FUNCTION_BLOCK TEMPLATE_NEURALFB
  (* Standard: 61499-2 *)
  (* Version 1.0, 11-01-12, GASR, Universidade do Estado de Santa Catarina *)
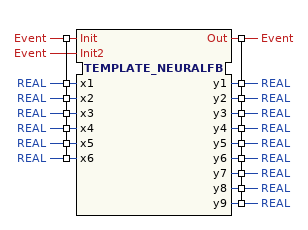
  EVENT_INPUT
    Init WITH x1, x2, x3, x4, x5, x6;
    Init2;
  END_EVENT
  EVENT_OUTPUT
    Out WITH y1, y2, y3, y4, y5, y6, y7, y8, y9;
  END_EVENT
  VAR_INPUT
    x1 : REAL;
    x2 : REAL;
    x3 : REAL;
    x4 : REAL;
    x5 : REAL;
    x6 : REAL;
  END_VAR
  VAR_OUTPUT
    y1 : REAL;
    y2 : REAL;
    y3 : REAL;
    y4 : REAL;
    y5 : REAL;
    y6 : REAL;
    y7 : REAL;
    y8 : REAL;
    y9 : REAL;
  END_VAR
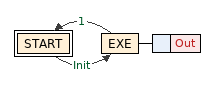
  EC_STATES
    START;
    EXE : -> Out;
  END_STATES
  EC_TRANSITIONS
    START TO EXE := Init;
    EXE TO START := 1;
  END_TRANSITIONS
END_FUNCTION_BLOCK
